PROGRAM PRG_Log_Main

VAR
	sysLogger 		: FB_SysLogLIstener;
	auditLogger		: FB_AuditLogLIstener;
END_VAR

sysLogger.CyclicLogic();
auditLogger.CyclicLogic();

END_PROGRAM

(* stored: Version 1.1.0.1
   POU PRG_Log_Main: Id {bb1d0e3f-e339-4d05-b071-4015d4af0ed5}, SpecialFunc None *)
